TYPE ST_CylinderX_HMI :
    STRUCT
        Config  : ST_Cylinder_Config;
        Command : ST_CylinderX_Command;
        Status  : ST_CylinderX_Status;
    END_STRUCT
END_TYPE

(* stored: Version 1.1.0.1
   DUT ST_CylinderX_HMI: Id {21cb6520-c345-430b-9d4d-d2bc0c55488f} *)
